TYPE "TMeasuring_Alarms"
VERSION : 0.1
// Block: TMeasuring_Alarms
   STRUCT
      TOMeasuring : Bool;
      MCFunction : Bool;
      TimeOutActivation : Bool;
   END_STRUCT;

END_TYPE
